// TIA Portal V20 export
// export: Created 2026-07-14T14:15:38.9498821Z, ExportSetting WithDefaults, DisplayName Totally Integrated Automation Portal, DisplayVersion V20 Update 5, DisplayName TIA Portal Openness, DisplayVersion V20 Update 4, DisplayName TIA Portal Version Control Interface, DisplayVersion V20 Update 5, DisplayName SINAMICS Startdrive Advanced, DisplayVersion V20, DisplayName SINAMICS DCC, DisplayVersion V20, DisplayName SINAMICS Startdrive G130, G150, S120, S150, SINAMICS MV, G220, S200, S210, DisplayVersion V20, DisplayName SINAMICS Startdrive G110M, G120, G120C, G120D, G120P, G115D, DisplayVersion V20, DisplayName STEP 7 Professional, DisplayVersion V20 Update 5, DisplayName STEP 7 Safety, DisplayVersion V20 Update 2, DisplayName WinCC Basic/Comfort/Advanced, DisplayVersion V20 Update 5, DisplayName WinCC Unified, DisplayVersion V20 Update 5
FUNCTION "BooleanExtras" : Void   // FC23, LAD
{ S7_Optimized_Access := 'TRUE' }
VERSION : 0.1
// Boolean reference examples (standalone Not, SCoil/RCoil)
// stored: AutoNumber true, IsIECCheckEnabled false, SetENOAutomatically false, UDAEnableTagReadback false
   VAR_TEMP
      EnableCmd : Bool;
      FaultLatch : Bool;
      RunA : Bool;
      StartCmd : Bool;
      Run : Bool;
      SetCmd : Bool;
      Motor1Latched : Bool;
      ResetCmd : Bool;
   END_VAR
BEGIN

REGION Network 1: Interlock inversion (Not)
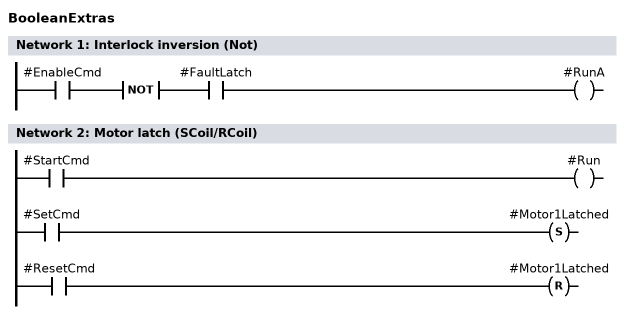
   RUNG wire#powerrail
      Contact( #EnableCmd )
      Not()
      Contact( #FaultLatch )
      Coil( #RunA )
   END_RUNG
   // the same network as SCL:
   #RunA := NOT #EnableCmd AND #FaultLatch;
END_REGION

REGION Network 2: Motor latch (SCoil/RCoil)
   RUNG wire#powerrail
      Contact( #StartCmd )
      Coil( #Run )
   END_RUNG
   RUNG wire#powerrail
      Contact( #SetCmd )
      S_Coil( #Motor1Latched )
   END_RUNG
   RUNG wire#powerrail
      Contact( #ResetCmd )
      R_Coil( #Motor1Latched )
   END_RUNG
   // the same network as SCL:
   #Run := #StartCmd;
   IF #SetCmd THEN #Motor1Latched := TRUE; END_IF;
   IF #ResetCmd THEN #Motor1Latched := FALSE; END_IF;
END_REGION
END_FUNCTION
